% RSLogix 500 project I2P JOB 13B - FORWARD-REVERSE USING 3 PBS OF 1P MOTOR_BAK026.RSS, saved by version 10.00.00.00 %
PROJECT "ML5B"    % processor: Bul.1763 MicroLogix 1100 Series B %

PROGRAM FILES
  LAD 2   14 rungs

DATA FILES
  O0 OUTPUT  4 elements
  I1 INPUT  6 elements
  S2 STATUS  66 elements
  B3 BINARY  2 elements
  T4 TIMER  1 elements
  C5 COUNTER  1 elements
  R6 CONTROL  1 elements
  N7 INTEGER  3 elements
  F8 FLOAT  1 elements

LADDER 2
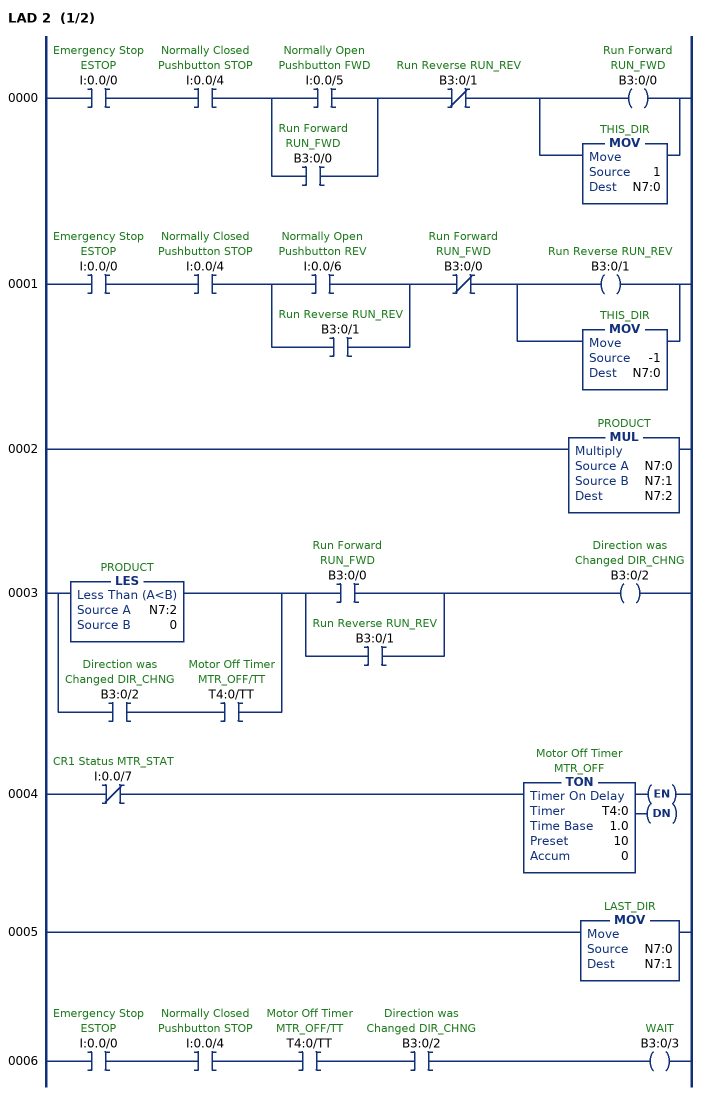
% Rung: 0 %
SOR XIC I:0.0/0 XIC I:0.0/4 BST XIC I:0.0/5 NXB XIC B3:0/0 BND XIO B3:0/1 BST OTE B3:0/0 NXB MOV 1 N7:0 BND EOR
%   I:0.0/0  ESTOP  "Emergency Stop" %
%   I:0.0/4  STOP  "Normally Closed Pushbutton" %
%   I:0.0/5  FWD  "Normally Open Pushbutton" %
%   B3:0/0  RUN_FWD  "Run Forward" %
%   B3:0/1  RUN_REV  "Run Reverse" %
%   N7:0  THIS_DIR %
% Rung: 1 %
SOR XIC I:0.0/0 XIC I:0.0/4 BST XIC I:0.0/6 NXB XIC B3:0/1 BND XIO B3:0/0 BST OTE B3:0/1 NXB MOV -1 N7:0 BND EOR
%   I:0.0/0  ESTOP  "Emergency Stop" %
%   I:0.0/4  STOP  "Normally Closed Pushbutton" %
%   I:0.0/6  REV  "Normally Open Pushbutton" %
%   B3:0/1  RUN_REV  "Run Reverse" %
%   B3:0/0  RUN_FWD  "Run Forward" %
%   N7:0  THIS_DIR %
% Rung: 2 %
SOR MUL N7:0 N7:1 N7:2 EOR
%   N7:0  THIS_DIR %
%   N7:1  LAST_DIR %
%   N7:2  PRODUCT %
% Rung: 3 %
SOR BST LES N7:2 0 NXB XIC B3:0/2 XIC T4:0/TT BND BST XIC B3:0/0 NXB XIC B3:0/1 BND OTE B3:0/2 EOR
%   N7:2  PRODUCT %
%   B3:0/2  DIR_CHNG  "Direction was Changed" %
%   T4:0  MTR_OFF  "Motor Off Timer" %
%   B3:0/0  RUN_FWD  "Run Forward" %
%   B3:0/1  RUN_REV  "Run Reverse" %
% Rung: 4 %
SOR XIO I:0.0/7 TON T4:0 1.0 10 0 EOR
%   I:0.0/7  MTR_STAT  "CR1 Status" %
%   T4:0  MTR_OFF  "Motor Off Timer" %
% Rung: 5 %
SOR MOV N7:0 N7:1 EOR
%   N7:0  THIS_DIR %
%   N7:1  LAST_DIR %
% Rung: 6 %
SOR XIC I:0.0/0 XIC I:0.0/4 XIC T4:0/TT XIC B3:0/2 OTE B3:0/3 EOR
%   I:0.0/0  ESTOP  "Emergency Stop" %
%   I:0.0/4  STOP  "Normally Closed Pushbutton" %
%   T4:0  MTR_OFF  "Motor Off Timer" %
%   B3:0/2  DIR_CHNG  "Direction was Changed" %
%   B3:0/3  WAIT %

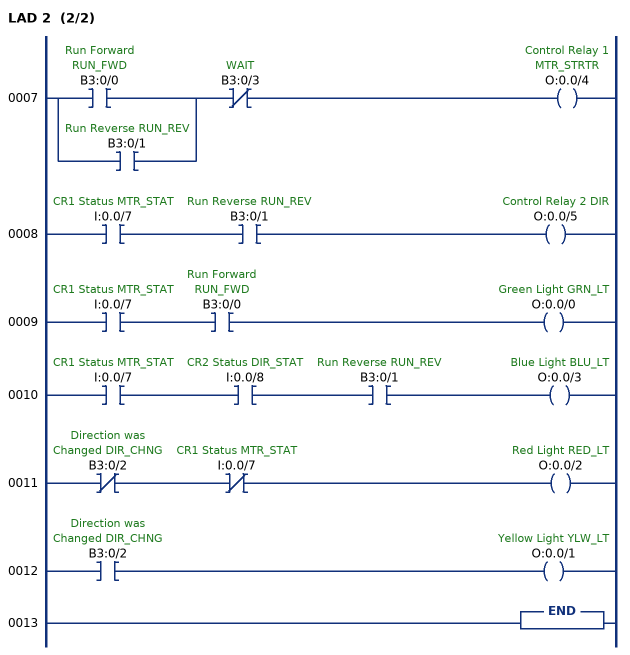
% Rung: 7 %
SOR BST XIC B3:0/0 NXB XIC B3:0/1 BND XIO B3:0/3 OTE O:0.0/4 EOR
%   B3:0/0  RUN_FWD  "Run Forward" %
%   B3:0/1  RUN_REV  "Run Reverse" %
%   B3:0/3  WAIT %
%   O:0.0/4  MTR_STRTR  "Control Relay 1" %
% Rung: 8 %
SOR XIC I:0.0/7 XIC B3:0/1 OTE O:0.0/5 EOR
%   I:0.0/7  MTR_STAT  "CR1 Status" %
%   B3:0/1  RUN_REV  "Run Reverse" %
%   O:0.0/5  DIR  "Control Relay 2" %
% Rung: 9 %
SOR XIC I:0.0/7 XIC B3:0/0 OTE O:0.0/0 EOR
%   I:0.0/7  MTR_STAT  "CR1 Status" %
%   B3:0/0  RUN_FWD  "Run Forward" %
%   O:0.0/0  GRN_LT  "Green Light" %
% Rung: 10 %
SOR XIC I:0.0/7 XIC I:0.0/8 XIC B3:0/1 OTE O:0.0/3 EOR
%   I:0.0/7  MTR_STAT  "CR1 Status" %
%   I:0.0/8  DIR_STAT  "CR2 Status" %
%   B3:0/1  RUN_REV  "Run Reverse" %
%   O:0.0/3  BLU_LT  "Blue Light" %
% Rung: 11 %
SOR XIO B3:0/2 XIO I:0.0/7 OTE O:0.0/2 EOR
%   B3:0/2  DIR_CHNG  "Direction was Changed" %
%   I:0.0/7  MTR_STAT  "CR1 Status" %
%   O:0.0/2  RED_LT  "Red Light" %
% Rung: 12 %
SOR XIC B3:0/2 OTE O:0.0/1 EOR
%   B3:0/2  DIR_CHNG  "Direction was Changed" %
%   O:0.0/1  YLW_LT  "Yellow Light" %
% Rung: 13 %
SOR END EOR

OTHER DOCUMENTED ADDRESSES
  I:0.0/1  3PSSA  "3 Position SS A"
  I:0.0/2  3PSSB  "3 Position SS B"
  I:0.0/3  2PSS  "2 Position SS"
  ONE  

DATA TABLE (non-zero values as saved)
DATA T4
% .PRE .ACC %
% T4:0 % 10 0
